FUNCTION_BLOCK HeartBeatBasic (* Basic Function Block Type *)
  (* Standard: 61499-2 *)
  (* Version 0.0, 7/17/2026, Schneider Electric, Template *)
  PACKAGE SE.Nereda;
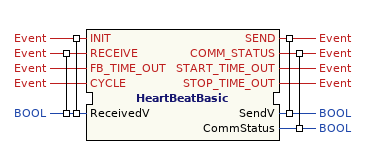
  EVENT_INPUT
    INIT WITH ReceivedV;
    RECEIVE WITH ReceivedV;
    FB_TIME_OUT;
    CYCLE;
  END_EVENT
  EVENT_OUTPUT
    SEND WITH SendV;
    COMM_STATUS WITH CommStatus;
    START_TIME_OUT;
    STOP_TIME_OUT;
  END_EVENT
  VAR_INPUT
    ReceivedV : BOOL;
  END_VAR
  VAR_OUTPUT
    SendV : BOOL;
    CommStatus : BOOL;
  END_VAR
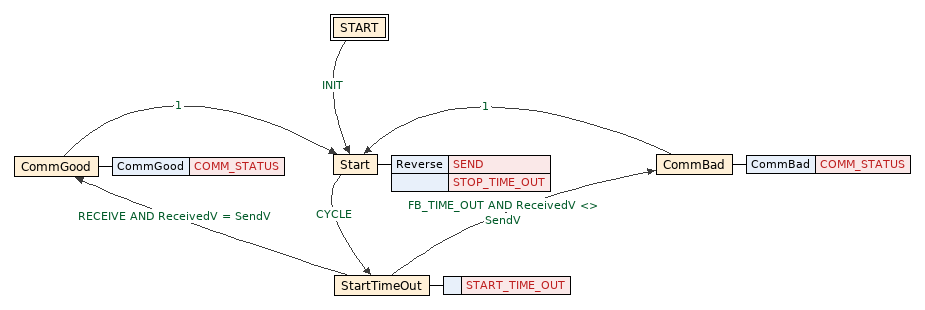
  EC_STATES
    START; (* Initial State *)
    Start : Reverse -> SEND, -> STOP_TIME_OUT;
    StartTimeOut : -> START_TIME_OUT;
    CommGood : CommGood -> COMM_STATUS;
    CommBad : CommBad -> COMM_STATUS;
  END_STATES
  EC_TRANSITIONS
    START TO Start := INIT;
    Start TO StartTimeOut := CYCLE;
    StartTimeOut TO CommGood := RECEIVE AND ReceivedV = SendV;
    CommGood TO Start := 1;
    StartTimeOut TO CommBad := FB_TIME_OUT AND ReceivedV <> SendV;
    CommBad TO Start := 1;
  END_TRANSITIONS
  ALGORITHM INIT IN ST: (* Initialization algorithm *)
;
  END_ALGORITHM
  ALGORITHM REQ IN ST: (* Normally executed algorithm *)
;
  END_ALGORITHM
  ALGORITHM Reverse IN ST:
;
SendV := NOT ReceivedV;
  END_ALGORITHM
  ALGORITHM CommGood IN ST:
;
CommStatus := TRUE;
  END_ALGORITHM
  ALGORITHM CommBad IN ST:
;
CommStatus := FALSE;
  END_ALGORITHM
END_FUNCTION_BLOCK
